INTERFACE I_SynchronousRpcHandler EXTENDS __SYSTEM.IQueryInterface

METHOD Handle
VAR_INPUT
	Parameters : I_Deserializer;
	Response : I_SynchronousRpcResponse;
END_VAR
END_METHOD

END_INTERFACE

(* stored: Version 1.1.0.1, ProductVersion 3.1.4024.12
   Itf I_SynchronousRpcHandler: Id {2a3870e6-6c22-0c53-3bfc-2541e1536c82}
   Method Handle: Id {71f049d1-00ad-0d90-1574-4cd39735e8f5} *)
